{attribute addProperty BoxType "EL3773-0000-0016"}
{attribute addProperty Id "I3_SAMPLESAT %I*ARRAY [1..10] OF INT16020"}
{attribute addProperty CRC "3386978351"}
{attribute addProperty SizeInBites "160"}
{attribute addProperty SizeInBytes "20"}
TYPE L3_Current_Samples_C9E1302F :
STRUCT
	{attribute addProperty Name "I3_SAMPLES"}
	I3_SAMPLES AT %I* : ARRAY [1..10] OF INT;
END_STRUCT
END_TYPE

(* stored: Version 1.2.0.0, ProductVersion 3.1.4024.9
   DUT L3_Current_Samples_C9E1302F: Id {c22cd9c3-94a5-4620-a5fb-a222ce7382d3} *)
